TYPE M1RadialSupportStatuses :
STRUCT
	///Operating status of the radial pressure setpoint
	pressureSetpointStatus: OperatingStatus;
	healthStatus: HealthStatus;
	busyStatus: BusyStatus;
END_STRUCT
END_TYPE

(* stored: Version 1.1.0.1, ProductVersion 3.1.4019.2
   DUT M1RadialSupportStatuses: Id {a5a294c0-f33c-4045-83a4-6d82147a27ce} *)
